Fanuc KAREL source: ka00091.KL

PROGRAM KA00091
%STACKSIZE=65535
%PRIORITY=65535
%NOLOCKGROUP
VAR
SRC : JOINTPOS9
DST : XYZWPREXT
BEGIN
-- UNSAFE_SOURCE_IR line 7: DST = convert_jointpos9_to_xyzwprext(SRC)
END KA00091
